RoboDK station: moving_object.rdk

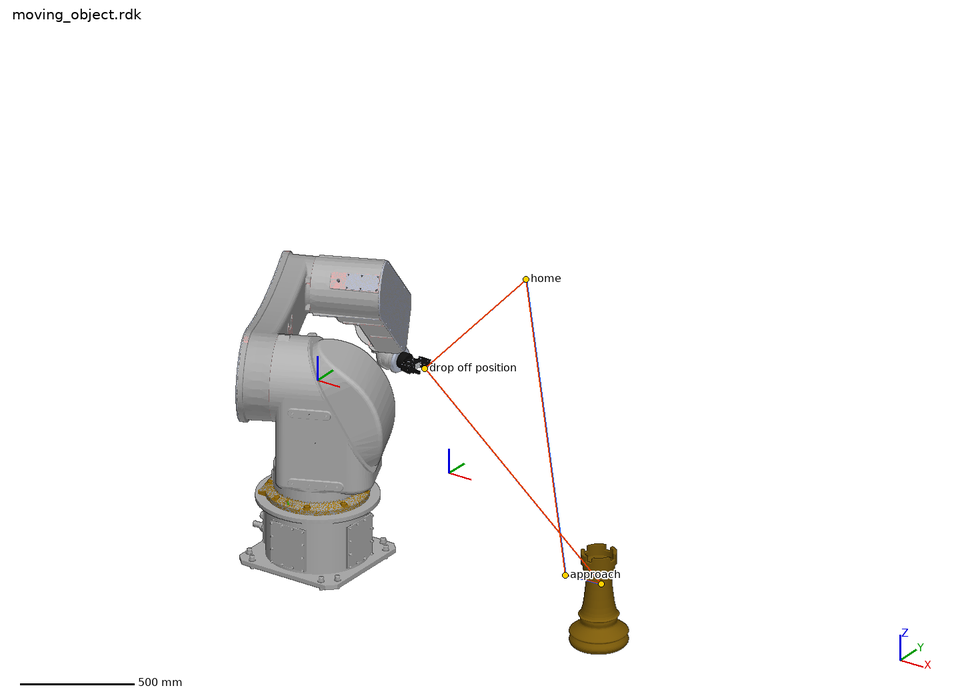
[picture v0: the station drawn from its stored meshes, robots at their saved joint values, targets as dots, program paths as lines]
Station moving_object (saved by RoboDK 5.5.4). Poses are relative to the parent item; angles as X-Y-Z fixed-axis rotations.
Station parameters (name, value as stored): LIN64
  - frame Fanuc P-50iB/10L Base at (0, 0, 850) mm
    - robot Fanuc P-50iB/10L: 6 axes, payload 10 kg, reach 1800 mm, repeatability 0.2 mm, weight 331 kg
        modified DH rows (alpha deg, a mm, theta deg, d mm): 0, 0, 0, 850; -90, 0, -90, 0; 0, 900, 0, 0; -90, 0, -90, 863.603; 70, 0, 0, 106.418; -70, 0, 0, 82
        base shift (0, 0, -850) mm
        joint limits [-160, -45, -205, -360, -360, -360] to [160, 120, 165, 360, 360, 360]; home [0, 0, 0, 0, 0, 0]; saved at [114.498, 88.832, -37.999, 12.076, -122.122, 84.343]
      - tool RobotiQ 2F-85 Gripper (Open), TCP at (0, 0, 130) mm, size 147.4 x 75 x 146.8 mm
  - frame Frame 2 at (0, 1000, 0) mm
    - target home (Cartesian target) at (1112, -1000, 1650) mm, rotated rx 0 ry -90 rz -180 deg; joints [0, 0, 0, 0, 0, 0] of Fanuc P-50iB/10L
    - target approach (Cartesian target) at (1320.42, -1000, 272.88) mm, rotated rx -87.55 ry -90 rz -92.45 deg; joints [5.081, 71.382, -75.011, 100.98, -80.836, -72.403] of Fanuc P-50iB/10L
    - target pickup position (Cartesian target) at (1498, -979.96, 271.41) mm, rotated rx 91.79 ry 4.66 rz 86.49 deg; joints [5.949, 75.329, -62.901, 91.574, -65.966, 22.142] of Fanuc P-50iB/10L
    - target drop off position (Cartesian target) at (-411.73, 404.55, 230.61) mm, rotated rx 91.79 ry 4.66 rz 86.49 deg; joints [114.498, 88.832, -37.999, 12.076, -122.122, 84.343] of Fanuc P-50iB/10L
  - program attach (1 instructions, listed below)
  - program dettach (1 instructions, listed below)
  - program move_rook_forward (9 instructions, listed below)
  - program move_rook_back (9 instructions, listed below)
  - program move_rook (3 instructions, listed below)
  - object Rook at (1500, 0, 0) mm, size 260.9 x 260.9 x 440 mm, geometry from Object Chess Rook.sld
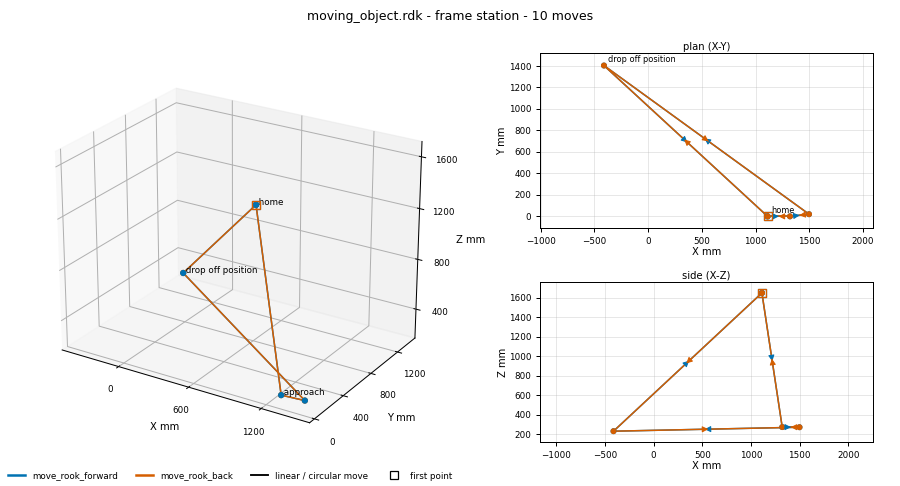
[picture p0: tool path of moving_object.rdk in frame station, 10 of 10 moves have a stored position in this frame; points joined in program order, loops and branches not executed]

--- program attach (robot Fanuc P-50iB/10L) ---
  Attach to RobotiQ 2F-85 Gripper (Open)

--- program dettach (robot Fanuc P-50iB/10L) ---
  Detach from RobotiQ 2F-85 Gripper (Open)

--- program move_rook_forward (robot Fanuc P-50iB/10L) ---
  Set Ref.: Frame 2
  Set Tool: RobotiQ 2F-85 Gripper (Open)
  MoveJ (home)
  MoveL (approach)
  MoveL (pickup position)
  Call attach
  MoveL (drop off position)
  Call dettach
  MoveL (home)

--- program move_rook_back (robot Fanuc P-50iB/10L) ---
  Set Ref.: Frame 2
  Set Tool: RobotiQ 2F-85 Gripper (Open)
  MoveJ (home)
  MoveL (drop off position)
  Call attach
  MoveL (pickup position)
  Call dettach
  MoveL (approach)
  MoveL (home)

--- program move_rook (robot Fanuc P-50iB/10L) ---
  Call move_rook_forward
  Pause 500 ms
  Call move_rook_back
